Fanuc KAREL source: CNV_STR_REAL.kl

PROGRAM T
%NOLOCKGROUP
VAR
 v0 : STRING[40]
 v1 : REAL
BEGIN
 CNV_STR_REAL(v0, v1)
END T
